FUNCTION_BLOCK Crane_PickUpWP EXTENDS ControlPrimitiveBase
VAR_INPUT
END_VAR
VAR_OUTPUT
END_VAR
VAR
	m_ptrCrane: POINTER TO Crane;
	
	m_step: INT := 0;
	m_timer: TON;
	
	// (EProcessVariables.Crane_HoldingWorkpiece = FALSE) AND (EProcessVariables.Crane_CylinderRetracted = TRUE)
	m_compExpr55: ComparisonExpression(EProcessVariables.Crane_HoldingWorkpiece, EComparisonType.equals, EDataType.binary, FALSE, 0, '', TRUE);
	m_compExpr57: ComparisonExpression(EProcessVariables.Crane_CylinderRetracted, EComparisonType.equals, EDataType.binary, TRUE, 0, '', TRUE);
	m_precondition: BoolExpression(m_compExpr55, EBoolOperation.and_op, m_compExpr57);
	
	// (EProcessVariables.Crane_HoldingWorkpiece = TRUE) AND (EProcessVariables.Crane_CylinderRetracted = TRUE)
	m_compExpr60: ComparisonExpression(EProcessVariables.Crane_HoldingWorkpiece, EComparisonType.equals, EDataType.binary, TRUE, 0, '', TRUE);
	m_compExpr62: ComparisonExpression(EProcessVariables.Crane_CylinderRetracted, EComparisonType.equals, EDataType.binary, TRUE, 0, '', TRUE);
	m_postcondition: BoolExpression(m_compExpr60, EBoolOperation.and_op, m_compExpr62);
END_VAR

SUPER^();

METHOD Abort : BOOL
VAR_INPUT
END_VAR
m_ptrCrane^.o_MonostableCylinder.METH_Retract();
IF m_ptrCrane^.o_VacuumGripper.WPTaken THEN
	m_ptrCrane^.o_VacuumGripper.METH_Intake();
ELSE
	m_ptrCrane^.o_VacuumGripper.METH_Release();
END_IF
Abort := TRUE;
END_METHOD

(* Execution logic of this Control Primitive. *)
METHOD PROTECTED  ExecuteInternal : BOOL
VAR_INPUT
	i_params: ParameterSet;
END_VAR
CASE m_step OF

	0:	// extend
		m_ptrCrane^.o_MonostableCylinder.METH_Extend();
		IF m_ptrCrane^.o_MonostableCylinder.Extended THEN
			m_step := 1;
		END_IF
	
	1:	// grip
		m_ptrCrane^.o_VacuumGripper.METH_Intake();
		m_timer(IN := TRUE, PT := T#1S);
		IF m_timer.Q THEN
			m_timer(IN := FALSE);
			m_step := 2;
		END_IF
	
	2:	// retract
		m_ptrCrane^.o_MonostableCylinder.METH_Retract();
		IF m_ptrCrane^.o_MonostableCylinder.Retracted THEN
			m_step := 0;
			ExecuteInternal := TRUE;
		END_IF	
END_CASE
END_METHOD

METHOD FB_init : BOOL
VAR_INPUT
	bInitRetains : BOOL; // if TRUE, the retain variables are initialized (warm start / cold start)
	bInCopyCode : BOOL;  // if TRUE, the instance afterwards gets moved into the copy code (online change)
	
	i_ptrCrane: POINTER TO Crane;
END_VAR
m_ptrCrane := i_ptrCrane;

m_id := EPrimitives.Crane_PickUpWP;
m_timeout := T#20S;

Precondition := m_precondition;
Postcondition := m_postcondition;
END_METHOD

END_FUNCTION_BLOCK

(* stored: Version 1.1.0.1, ProductVersion 3.1.4024.9
   POU Crane_PickUpWP: Id {c6ee90db-10e5-4113-a0c3-db35ef248192}, SpecialFunc None
   Method Abort: Id {50072af3-d62e-4a70-9b25-f213f2be3b99}
   Method ExecuteInternal: Id {c86ef8f0-fe75-45e9-a32a-7c4c49e828ec}
   Method FB_init: Id {2e89f0b2-f1d6-4d93-afa1-07c4c7e0d1fa} *)
